(* Schneider Machine Expert - Basic project Pollas, file version 2.7.0.0 *)
(* ProjectInformations: Name=Nuevo proyecto *)

HARDWARE
  Cpu 0: TM221CE40R
  EthernetConfiguration: NetworkName=M221, IpAllocationMode=FixedAddress, IpAddress=0.0.0.0, SubnetMask=0.0.0.0
  SerialLineConfiguration: Baud=Baud19200, Parity=ParityEven, DataBits=DataBits8, StopBits=StopBits1, PhysicalMedium=PhysicalMediumRs485, TransmissionMode=TransmissionModeModbusRtu, SlaveId=1, Addressing=SlaveAddressing
  MastTask: UsePeriodScanMode=false, PeriodScan=100
  FastTask: Period=255
  CpuBehavior: StartingMode=StartAsPreviousState, AutoSaveRamOnEeprom=true, WatchdogPeriod=250

SYMBOLS  (address, symbol, comment, settings)
  %TM0        [Preset=1]

POU Nuevo POU
  (* SectionNumber=1 *)

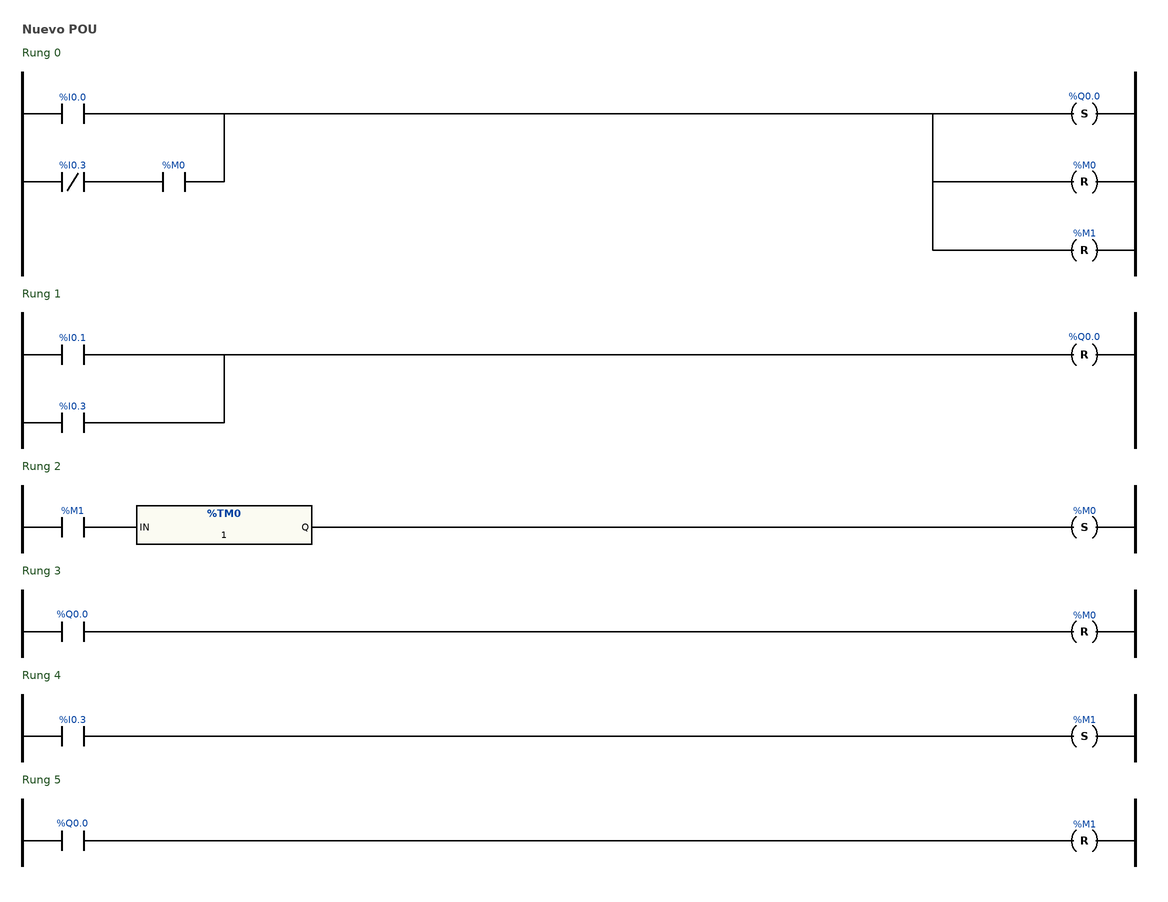

// Rung 0
  LD %I0.0
  OR(N %I0.3
  AND %M0
  )
  S %Q0.0
  R %M0
  R %M1
  // as ST:
  //   IF %I0.0 OR NOT %I0.3 AND %M0 THEN %Q0.0 := TRUE; END_IF;
  //   _t1 := %I0.0 OR NOT %I0.3 AND %M0;
  //   IF _t1 THEN %M0 := FALSE; END_IF;
  //   IF _t1 THEN %M1 := FALSE; END_IF;

// Rung 1
  LD %I0.1
  OR %I0.3
  R %Q0.0
  // as ST:
  //   IF %I0.1 OR %I0.3 THEN %Q0.0 := FALSE; END_IF;

// Rung 2
  BLK %TM0
  LD %M1
  IN
  OUT_BLK
  LD Q
  S %M0
  END_BLK
  // as ST:
  //   %TM0(IN := %M1);
  //   IF %TM0.Q THEN %M0 := TRUE; END_IF;

// Rung 3
  LD %Q0.0
  R %M0
  // as ST:
  //   IF %Q0.0 THEN %M0 := FALSE; END_IF;

// Rung 4
  LD %I0.3
  S %M1
  // as ST:
  //   IF %I0.3 THEN %M1 := TRUE; END_IF;

// Rung 5
  LD %Q0.0
  R %M1
  // as ST:
  //   IF %Q0.0 THEN %M1 := FALSE; END_IF;
